Yaskawa INFORM job: TWIN_FRONT_SEARCH_-90ST-1_5340.JBI

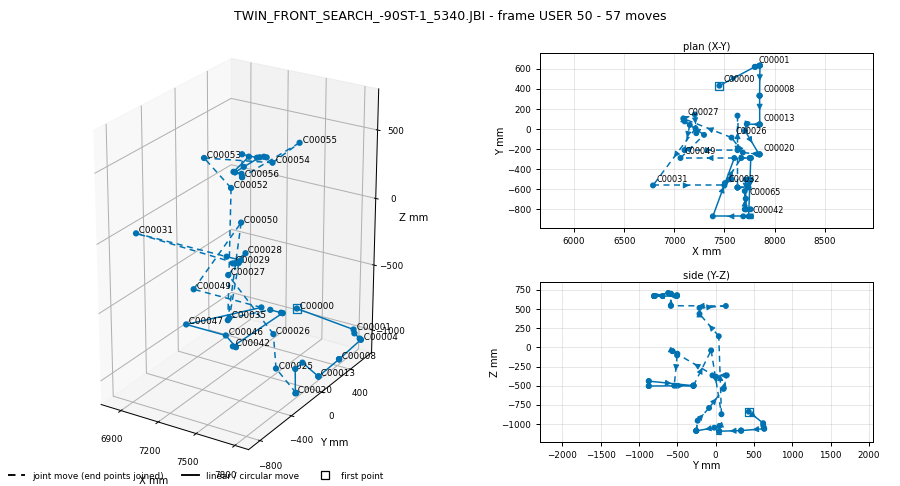
[picture p0: tool path of TWIN_FRONT_SEARCH_-90ST-1_5340.JBI in frame USER 50, 57 of 61 moves have a stored position in this frame; points joined in program order, loops and branches not executed]
/JOB
//NAME TWIN_FRONT_SEARCH_-90ST-1_5340
///FOLDERNAME 02-SKRZYNIE_JOBS
//POS
///NPOS 73,73,0,10,0,0
///USER 50
///TOOL 0
///POSTYPE USER
///RECTAN
///RCONF 1,0,0,0,0,0,0,0,0,0,0,0,0,0,0,0,0,0,0,0,0,0,0,0
C00000=7449.693,432.672,-838.681,56.3065,47.9522,-54.8413
///RCONF 0,0,0,0,0,0,0,0,0,0,0,0,0,0,0,0,0,0,0,0,0,0,0,0
C00001=7802.169,620.288,-988.612,32.6060,47.2119,-72.4114
C00002=7808.739,621.464,-1017.218,32.8145,47.1981,-91.3467
C00003=7846.524,631.738,-1052.508,32.8164,47.1964,-91.3435
C00004=7854.677,633.926,-1060.092,32.8170,47.1961,-91.3442
C00005=7854.715,633.894,-1071.517,32.8197,47.1956,-91.3440
C00006=7866.908,633.931,-1068.545,32.8156,47.1972,-91.3457
C00007=7854.677,633.926,-1060.092,32.8170,47.1961,-91.3442
///RCONF 1,0,0,0,0,0,0,0,0,0,0,0,0,0,0,0,0,0,0,0,0,0,0,0
C00008=7850.902,332.846,-1085.287,31.8440,42.1242,-91.3303
C00009=7850.902,332.846,-1085.287,31.8440,42.1242,-91.3303
C00010=7850.895,332.850,-1091.855,31.8451,42.0926,-91.3273
C00011=7864.909,332.841,-1088.803,31.8466,42.0967,-91.3338
C00012=7850.902,332.846,-1085.287,31.8440,42.1242,-91.3303
C00013=7852.585,46.085,-1092.978,31.8356,42.1288,-99.9874
C00014=7852.585,46.085,-1092.978,31.8356,42.1288,-99.9874
C00015=7852.594,46.067,-1101.750,31.8361,42.1281,-99.9887
C00016=7864.183,46.071,-1098.714,31.8368,42.1302,-99.9918
C00017=7852.585,46.085,-1092.978,31.8356,42.1288,-99.9874
///RCONF 0,0,0,0,0,0,0,0,0,0,0,0,0,0,0,0,0,0,0,0,0,0,0,0
C00018=7723.295,49.630,-1023.685,34.3031,14.5531,-54.8249
C00019=7706.141,-17.501,-1047.481,-6.2879,-10.7592,27.7896
///RCONF 1,0,0,0,0,0,0,0,0,0,0,0,0,0,0,0,0,0,0,0,0,0,0,0
C00020=7848.205,-254.977,-1089.028,-23.4725,44.5717,116.2705
C00021=7852.206,-251.604,-1086.783,-23.4742,44.5702,116.2668
C00022=7852.193,-251.597,-1096.561,-23.4742,44.5690,116.2657
C00023=7862.735,-251.605,-1093.564,-23.4733,44.5682,116.2640
C00024=7852.206,-251.604,-1086.783,-23.4742,44.5702,116.2668
C00025=7683.234,-234.173,-956.259,-23.4688,44.5707,116.2734
C00026=7570.999,-84.978,-789.821,-8.3295,54.7414,178.0447
C00027=7089.632,105.235,-540.772,34.6747,-14.1850,-36.1511
///RCONF 0,0,0,0,0,0,0,0,0,0,0,0,0,0,0,0,0,0,0,0,0,0,0,0
C00028=7204.424,145.895,-364.343,71.1061,41.6311,-75.1821
C00029=7219.459,-40.999,-365.280,-52.3016,-20.5804,53.0667
C00030=7211.681,7.015,-383.291,11.0196,-43.7028,-11.2189
///RCONF 1,0,1,0,0,0,0,0,0,0,0,0,0,0,0,0,0,0,0,0,0,0,0,0
C00031=6787.828,-561.979,-49.248,-84.3346,30.5101,20.5434
///RCONF 0,0,1,0,1,0,0,0,0,0,0,0,0,0,0,0,0,0,0,0,0,0,0,0
C00032=7499.847,-561.979,-49.248,-84.3345,30.5096,20.5433
///RCONF 0,0,1,0,0,0,0,0,0,0,0,0,0,0,0,0,0,0,0,0,0,0,0,0
C00033=7568.245,-498.271,-82.797,69.9077,-7.2021,-117.4885
C00034=7554.743,-500.998,-104.255,54.0039,-31.4868,-103.9439
///RCONF 0,0,0,0,0,0,0,0,0,0,0,0,0,0,0,0,0,0,0,0,0,0,0,0
C00035=7504.887,-539.129,-499.841,26.1477,-33.6094,-90.8544
C00036=7668.096,-288.720,-499.869,26.1496,-33.6072,-90.8555
C00037=7751.665,-288.695,-499.888,50.2103,-29.8101,-103.4316
C00038=7768.930,-288.682,-499.895,50.2097,-29.8104,-103.4300
C00039=7763.119,-288.672,-499.903,50.1917,-29.7456,-103.4205
C00040=7763.103,-288.680,-520.622,50.1900,-29.7472,-103.4203
C00041=7763.119,-288.672,-499.903,50.1917,-29.7456,-103.4205
C00042=7741.293,-870.810,-504.158,50.1892,-29.7500,-103.4230
C00043=7771.566,-870.808,-504.148,50.1915,-29.7488,-103.4245
C00044=7764.374,-870.799,-504.146,50.1908,-29.7492,-103.4235
C00045=7765.764,-870.775,-524.906,50.1908,-29.7505,-103.4216
C00046=7687.703,-870.770,-440.257,50.1921,-29.7495,-103.4228
C00047=7384.219,-870.770,-440.257,50.1921,-29.7495,-103.4228
C00048=7598.862,-288.695,-499.888,50.2103,-29.8101,-103.4316
C00049=7061.929,-288.695,-499.888,50.2103,-29.8101,-103.4316
C00050=7296.409,-57.933,-39.561,132.2856,-81.6072,-138.1355
C00051=7103.855,76.465,-871.663,11.0010,-20.3154,-11.3718
///RCONF 1,0,1,0,0,0,0,0,0,0,0,0,0,0,0,0,0,0,0,0,0,0,0,0
C00052=7154.189,41.489,145.490,17.6136,-33.4406,-10.5318
C00053=7102.089,-209.900,436.597,-19.7303,-44.5925,9.1969
C00054=7630.528,-209.897,514.987,-19.7320,-44.5912,9.1993
C00055=7630.528,133.977,539.739,-61.9423,-30.0021,35.7336
C00056=7630.500,-582.850,542.955,-61.9434,-30.0005,35.7331
C00057=7630.491,-582.857,542.952,-61.9449,-29.9979,35.7338
C00058=7630.501,-582.856,698.927,-61.9436,-29.9977,35.7338
C00059=7740.859,-582.856,698.927,-61.9436,-29.9977,35.7338
C00060=7743.607,-503.312,679.062,-61.9419,-29.9985,35.7328
C00061=7767.014,-503.295,679.048,-61.9411,-29.9999,35.7333
C00062=7763.629,-503.296,679.051,-61.9419,-29.9991,35.7339
C00063=7763.591,-503.318,652.327,-61.9418,-30.0006,35.7318
C00064=7712.855,-503.315,668.869,-61.9405,-30.0044,35.7306
C00065=7712.852,-694.511,668.854,-61.9406,-30.0033,35.7302
C00066=7713.637,-800.128,668.857,-61.9367,-30.0090,35.7263
C00067=7713.637,-800.128,668.857,-61.9367,-30.0090,35.7263
C00068=7766.968,-800.141,668.851,-61.9359,-30.0085,35.7248
C00069=7762.089,-800.140,668.843,-61.9353,-30.0078,35.7247
C00070=7762.089,-800.143,652.075,-61.9332,-30.0093,35.7234
C00071=7703.046,-800.145,669.668,-61.9339,-30.0066,35.7239
C00072=7703.033,-618.392,709.694,-61.9347,-30.0087,35.7238
///RCONF 0,0,0,0,0,0,0,0,0,0,0,0,0,0,0,0,0,0,0,0,0,0,0,0
BC00000=5892.685
BC00001=6515.049
BC00002=6515.049
BC00003=6515.049
BC00004=6515.049
BC00005=6515.049
BC00006=6515.049
BC00007=6515.049
BC00008=6515.055
BC00009=6515.055
BC00010=6515.055
BC00011=6515.055
BC00012=6515.055
BC00013=6515.049
BC00014=6515.049
BC00015=6515.049
BC00016=6515.049
BC00017=6515.049
BC00018=6515.049
BC00019=6515.049
BC00020=6515.049
BC00021=6515.049
BC00022=6515.049
BC00023=6515.049
BC00024=6515.049
BC00025=6428.036
BC00026=6132.885
BC00027=5388.459
BC00028=5388.459
BC00029=5388.459
BC00030=5388.459
BC00031=5388.459
BC00032=6100.478
BC00033=6100.478
BC00034=6100.478
BC00035=6331.805
BC00036=6331.805
BC00037=6331.805
BC00038=6331.805
BC00039=6331.805
BC00040=6331.805
BC00041=6331.805
BC00042=6331.805
BC00043=6331.805
BC00044=6331.805
BC00045=6331.805
BC00046=6331.805
BC00047=6028.321
BC00048=6179.002
BC00049=5642.069
BC00050=5642.069
BC00051=5642.069
BC00052=5642.069
BC00053=5642.069
BC00054=6170.513
BC00055=6170.513
BC00056=6170.513
BC00057=6302.692
BC00058=6302.692
BC00059=6413.050
BC00060=6413.050
BC00061=6413.050
BC00062=6413.050
BC00063=6413.050
BC00064=6413.050
BC00065=6556.947
BC00066=6565.475
BC00067=6565.475
BC00068=6565.475
BC00069=6565.475
BC00070=6565.475
BC00071=6565.475
BC00072=6565.475
///POSTYPE BASE
P00006=-2.449,0.031,8.825,0.0000,0.0000,0.0000
P00021=6.550,-0.003,-5.735,0.0000,0.0000,0.0000
P00022=5.943,-0.018,-6.388,0.0000,0.0000,0.0000
P00023=7.025,-0.019,-7.168,0.0000,0.0000,0.0000
P00024=5.926,-0.047,-4.777,0.0000,0.0000,0.0000
P00058=0.000,0.000,3.000,0.0000,0.0000,0.0000
P00501=-2.026,0.009,3.534,0.0000,0.0000,0.0000
///RCONF 1,0,0,0,0,0,0,0,0,0,0,0,0,0,0,0,0,0,0,0,0,0,0,0
P00502=-2.023,0.001,1.732,0.0000,0.0000,0.0000
P00503=0.138,-0.044,1.539,0.0000,0.0000,0.0000
P00504=-0.309,-0.010,1.636,0.0000,0.0000,0.0000
//INST
///DATE 2024/10/28 14:47
///ATTR SC,RW,RJ
////FRAME USER 50
///GROUP1 RB1,BS1
NOP
MOVJ C00000 BC00000 VJ=40.00
'::::::::::::::::::::::::::::::::
'W56 P
'::::::::::::::::::::::::::::::::
MOVL C00001 BC00001 V=500.0
MOVL C00002 BC00002 V=500.0
MOVL C00003 BC00003 V=500.0
MOVL C00004 BC00004 V=166.7 PL=0
REFP 3 C00005 BC00005
CALL JOB:SEARCH-R1
IMOV P0058 V=23.0
SET P0501 P0006
SFTON P0501
REFP 3 C00006 BC00006
CALL JOB:SEARCH-R1
SET P0501 P0006
SFTON P0501
MOVL C00007 BC00007 V=166.7 PL=0
SFTOF
'::::::::::::::::::::::::::::::::
'W56 L
'::::::::::::::::::::::::::::::::
MOVL C00008 BC00008 V=333.3
MOVL C00009 BC00009 V=166.7 PL=0
REFP 3 C00010 BC00010
CALL JOB:SEARCH-R1
IMOV P0058 V=23.0
SET P0502 P0006
SFTON P0502
REFP 3 C00011 BC00011
CALL JOB:SEARCH-R1
SET P0502 P0006
SFTON P0502
MOVL C00012 BC00012 V=166.7 PL=0
SFTOF
'::::::::::::::::::::::::::::::::
'W57 P
'::::::::::::::::::::::::::::::::
MOVL C00013 BC00013 V=250.0
MOVL C00014 BC00014 V=166.7 PL=0
REFP 3 C00015 BC00015
CALL JOB:SEARCH-R1
IMOV P0058 V=23.0
SET P0503 P0006
SFTON P0503
REFP 3 C00016 BC00016
CALL JOB:SEARCH-R1
SET P0503 P0006
SFTON P0503
MOVL C00017 BC00017 V=250.0 PL=0
SFTOF
'::::::::::::::::::::::::::::::::
'W57 L
'::::::::::::::::::::::::::::::::
MOVL C00018 BC00018 V=333.3
MOVL C00019 BC00019 V=333.3
MOVL C00020 BC00020 V=333.3
MOVL C00021 BC00021 V=166.7 PL=0
REFP 3 C00022 BC00022
CALL JOB:SEARCH-R1
IMOV P0058 V=23.0
SET P0504 P0006
SFTON P0504
REFP 3 C00023 BC00023
CALL JOB:SEARCH-R1
SET P0504 P0006
SFTON P0504
MOVL C00024 BC00024 V=166.7 PL=0
SFTOF
MOVJ C00025 BC00025 VJ=40.00
MOVJ C00026 BC00026 VJ=50.00
MOVJ C00027 BC00027 VJ=50.00
MOVJ C00028 BC00028 VJ=50.00
MOVJ C00029 BC00029 VJ=50.00
MOVJ C00030 BC00030 VJ=50.00
MOVJ C00031 BC00031 VJ=50.00
MOVJ C00032 BC00032 VJ=50.00
MOVL C00033 BC00033 V=166.7
MOVJ C00034 BC00034 VJ=50.00
MOVJ C00035 BC00035 VJ=50.00
MOVJ C00036 BC00036 VJ=50.00
MOVL C00037 BC00037 V=166.7
REFP 3 C00038 BC00038
CALL JOB:SEARCH-R1
SET P0021 P0006
SFTON P0021
MOVL C00039 BC00039 V=166.7 PL=0
REFP 3 C00040 BC00040
CALL JOB:SEARCH-R1
SET P0021 P0006
SFTON P0021
MOVL C00041 BC00041 V=166.7 PL=0
SFTOF
MOVL C00042 BC00042 V=166.7
REFP 3 C00043 BC00043
CALL JOB:SEARCH-R1
SET P0022 P0006
SFTON P0022
MOVL C00044 BC00044 V=166.7 PL=0
REFP 3 C00045 BC00045
CALL JOB:SEARCH-R1
SET P0022 P0006
SFTON P0022
MOVL C00046 BC00046 V=166.7 PL=0
MOVL C00047 BC00047 V=166.7
SFTOF
MOVL C00048 BC00048 V=166.7
MOVJ C00049 BC00049 VJ=50.00
MOVJ C00050 BC00050 VJ=50.00
MOVJ C00051 BC00051 VJ=50.00
MOVJ C00052 BC00052 VJ=50.00
MOVJ C00053 BC00053 VJ=50.00
MOVJ C00054 BC00054 VJ=50.00
MOVJ C00055 BC00055 VJ=50.00
MOVJ C00056 BC00056 VJ=50.00
MOVJ C00057 BC00057 VJ=50.00
MOVJ C00058 BC00058 VJ=50.00
MOVL C00059 BC00059 V=166.7
MOVL C00060 BC00060 V=166.7
REFP 3 C00061 BC00061
CALL JOB:SEARCH-R1
SET P0023 P0006
SFTON P0023
MOVL C00062 BC00062 V=166.7 PL=0
REFP 3 C00063 BC00063
CALL JOB:SEARCH-R1
SET P0023 P0006
SFTON P0023
MOVL C00064 BC00064 V=166.7 PL=0
MOVL C00065 BC00065 V=166.7
SFTOF
MOVL C00066 BC00066 V=166.7
MOVL C00067 BC00067 V=166.7
REFP 3 C00068 BC00068
CALL JOB:SEARCH-R1
SET P0024 P0006
SFTON P0024
MOVL C00069 BC00069 V=166.7 PL=0
REFP 3 C00070 BC00070
CALL JOB:SEARCH-R1
SET P0024 P0006
SFTON P0024
MOVL C00071 BC00071 V=166.7 PL=0
MOVL C00072 BC00072 V=166.7
SFTOF
END
